FUNCTION_BLOCK ArrayMulCumulative_Real5 (* Basic FB with empty ECC *)
  (* Standard: 61499-2 *)
  (* Version 1.0, 2020-08-15, Candra Wardaya, UGM *)
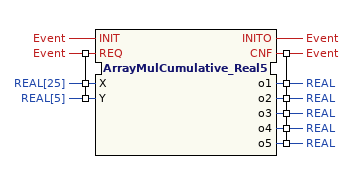
  EVENT_INPUT
    INIT;
    REQ WITH X, Y;
  END_EVENT
  EVENT_OUTPUT
    INITO;
    CNF WITH o1, o2, o3, o4, o5;
  END_EVENT
  VAR_INPUT
    X : ARRAY [0..24] OF REAL;
    Y : ARRAY [0..4] OF REAL;
  END_VAR
  VAR_OUTPUT
    o1 : REAL;
    o2 : REAL;
    o3 : REAL;
    o4 : REAL;
    o5 : REAL;
  END_VAR
  VAR
    i : INT; (* Internal Variable *)
    val1 : REAL; (* Internal Variable *)
  END_VAR
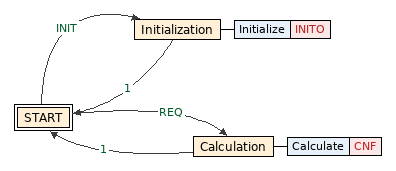
  EC_STATES
    START; (* Initial State *)
    Initialization : Initialize -> INITO;
    Calculation : Calculate -> CNF;
  END_STATES
  EC_TRANSITIONS
    START TO Initialization := INIT;
    Initialization TO START := 1;
    START TO Calculation := REQ;
    Calculation TO START := 1;
  END_TRANSITIONS
  ALGORITHM Initialize IN ST: (* New Algorithm *)

  END_ALGORITHM
  ALGORITHM Calculate IN ST: (* New Algorithm *)
o1 := X[0]*Y[0] + X[1]*Y[1] + X[2]*Y[2] + X[3]*Y[3] + X[4]*Y[4] ;
o2 := X[5]*Y[0] + X[6]*Y[1] + X[7]*Y[2] + X[8]*Y[3] + X[9]*Y[4] ;
o3 := X[10]*Y[0] + X[11]*Y[1] + X[12]*Y[2] + X[13]*Y[3] + X[14]*Y[4] ;
o4 := X[15]*Y[0] + X[16]*Y[1] + X[17]*Y[2] + X[18]*Y[3] + X[19]*Y[4] ;
o5 := X[20]*Y[0] + X[21]*Y[1] + X[22]*Y[2] + X[23]*Y[3] + X[24]*Y[4] ;
  END_ALGORITHM
END_FUNCTION_BLOCK
